// TIA Portal V18 export
FUNCTION "ST10Cyl_interface81-90" : Void   // FC1028, LAD
{ S7_Optimized_Access := 'FALSE' }
VERSION : 0.1
// stored: AutoNumber false, IsIECCheckEnabled false, SetENOAutomatically false, UDAEnableTagReadback false
   VAR_INPUT
      AlwaysON : Bool;
      E_stop : Bool;
   END_VAR
   VAR_TEMP
      tTest : Bool;
   END_VAR
BEGIN

REGION Network 1 (SCL): Cylinder 81-90 IO Interface (SCL)
   (*
   //Cylinder81 IO  L-UnloadingTransCylinder
   //Input
   "ST10Cylinder".Cy[81].In.WorkPositionSensor := "iL-UnloadingTransCylinderInWP";
   "ST10Cylinder".Cy[81].In.HomePositionSensor := "iL-UnloadingTransCylinderInHP";
   //Output
   "oL-UnloadingTransCylinderToWP" := "ST10Cylinder".Cy[81].Out.GoWorkPosition;
   "oL-UnloadingTransCylinderToHP" := "ST10Cylinder".Cy[81].Out.GoHomePosition;

   //Cylinder82 IO  L-UnloadingTransPalletLocationCylinder
   //Input
   "ST10Cylinder".Cy[82].In.WorkPositionSensor := "iL-UnloadingTransPalletLocationCylinderInWP";
   "ST10Cylinder".Cy[82].In.HomePositionSensor := "iL-UnloadingTransPalletLocationCylinderInHP";
   //Output
   "oL-UnloadingTransPalletLocationCylinderToWP" := "ST10Cylinder".Cy[82].Out.GoWorkPosition;
   "oL-UnloadingTransPalletLocationCylinderToHP" := "ST10Cylinder".Cy[82].Out.GoHomePosition;

   //Cylinder83 IO  L-UnloadingStopperCylinder1_1
   //Input
   "ST10Cylinder".Cy[83].In.WorkPositionSensor := "oL-UnloadingStopperCylinder1_1";
   "ST10Cylinder".Cy[83].In.HomePositionSensor := NOT "oL-UnloadingStopperCylinder1_1";
   //Output
   "oL-UnloadingStopperCylinder1_1" := "ST10Cylinder".Cy[83].Out.GoWorkPosition;
   //"oI-0030TrayLoading8trayStopperCylinderToHP" := "ST10Cylinder".Cy[83].Out.GoHomePosition;

   //Cylinder84 IO  L-UnloadingStopperCylinder1_2
   //Input
   "ST10Cylinder".Cy[84].In.WorkPositionSensor := "oL-UnloadingStopperCylinder1_2";
   "ST10Cylinder".Cy[84].In.HomePositionSensor := NOT "oL-UnloadingStopperCylinder1_2";
   //Output
   "oL-UnloadingStopperCylinder1_2" := "ST10Cylinder".Cy[84].Out.GoWorkPosition;
   //"oI-0080TrayLoadingTaketrayCylinderToHP" := "ST10Cylinder".Cy[84].Out.GoHomePosition;

   //Cylinder85 IO  L-UnloadingStopperCylinder2_1
   //Input
   "ST10Cylinder".Cy[85].In.WorkPositionSensor := "oL-UnloadingStopperCylinder2_1";
   "ST10Cylinder".Cy[85].In.HomePositionSensor := NOT "oL-UnloadingStopperCylinder2_1";
   //Output
   "oL-UnloadingStopperCylinder2_1" := "ST10Cylinder".Cy[85].Out.GoWorkPosition;
   //"oI-0050TrayLoadingTrayCylinderToHP" := "ST10Cylinder".Cy[85].Out.GoHomePosition;

   //Cylinder86  L-UnloadingStopperCylinder2_2
   //Input
   "ST10Cylinder".Cy[86].In.WorkPositionSensor := "oL-UnloadingStopperCylinder2_2";
   "ST10Cylinder".Cy[86].In.HomePositionSensor := NOT "oL-UnloadingStopperCylinder2_2";
   //Output
   "oL-UnloadingStopperCylinder2_2" := "ST10Cylinder".Cy[86].Out.GoWorkPosition;
   //"oI-0080TrayLoadingTraySupportCylinder1ToHP" := "ST10Cylinder".Cy[86].Out.GoHomePosition;

   //Cylinder87 L-UnloadingStopperCylinder3_1
   //Input
   "ST10Cylinder".Cy[87].In.WorkPositionSensor := "oL-UnloadingStopperCylinder3_1";
   "ST10Cylinder".Cy[87].In.HomePositionSensor := NOT "oL-UnloadingStopperCylinder3_1";
   //Output
   "oL-UnloadingStopperCylinder3_1" := "ST10Cylinder".Cy[87].Out.GoWorkPosition;
   //"oI-0070TrayLoadingTraySupportCylinder8ToHP" := "ST10Cylinder".Cy[87].Out.GoHomePosition;

   //Cylinder88 L-UnloadingStopperCylinder3_2
   //Input
   "ST10Cylinder".Cy[88].In.WorkPositionSensor := "oL-UnloadingStopperCylinder3_2";
   "ST10Cylinder".Cy[88].In.HomePositionSensor := NOT "oL-UnloadingStopperCylinder3_2";
   //Output
   "oL-UnloadingStopperCylinder3_2" := "ST10Cylinder".Cy[88].Out.GoWorkPosition;
   //"oI-0080TrayLoadingTrayLocationCylinderToHP" := "ST10Cylinder".Cy[88].Out.GoHomePosition;
   //
   *)
   (*
   //Cylinder89 K-reserveLoadingStopperCylinder4_1
   //Input
   "ST10Cylinder".Cy[89].In.WorkPositionSensor := "oK-reserveLoadingStopperCylinder4_1";
   "ST10Cylinder".Cy[89].In.HomePositionSensor := NOT "oK-reserveLoadingStopperCylinder4_1";
   //Output
   "oK-reserveLoadingStopperCylinder4_1" := "ST10Cylinder".Cy[89].Out.GoWorkPosition;
   //"oI-0090TrayLoadingTrayUnloadingLiftingCylinderToHP" := "ST10Cylinder".Cy[89].Out.GoHomePosition;

   //Cylinder70 K-reserveLoadingStopperCylinder4_2
   // //Input
   "ST10Cylinder".Cy[70].In.WorkPositionSensor := "oK-reserveLoadingStopperCylinder4_2";
   "ST10Cylinder".Cy[70].In.HomePositionSensor := NOT "oK-reserveLoadingStopperCylinder4_2";
   // //Output
   "oK-reserveLoadingStopperCylinder4_2" := "ST10Cylinder".Cy[70].Out.GoWorkPosition;
   // "Feeding washer  lift Cylinder ToHP" := "ST10Cylinder".Cy[70].Out.GoHomePosition;

   *)
END_REGION

REGION Network 2: CY81 interface L-UnloadingTransCylinder
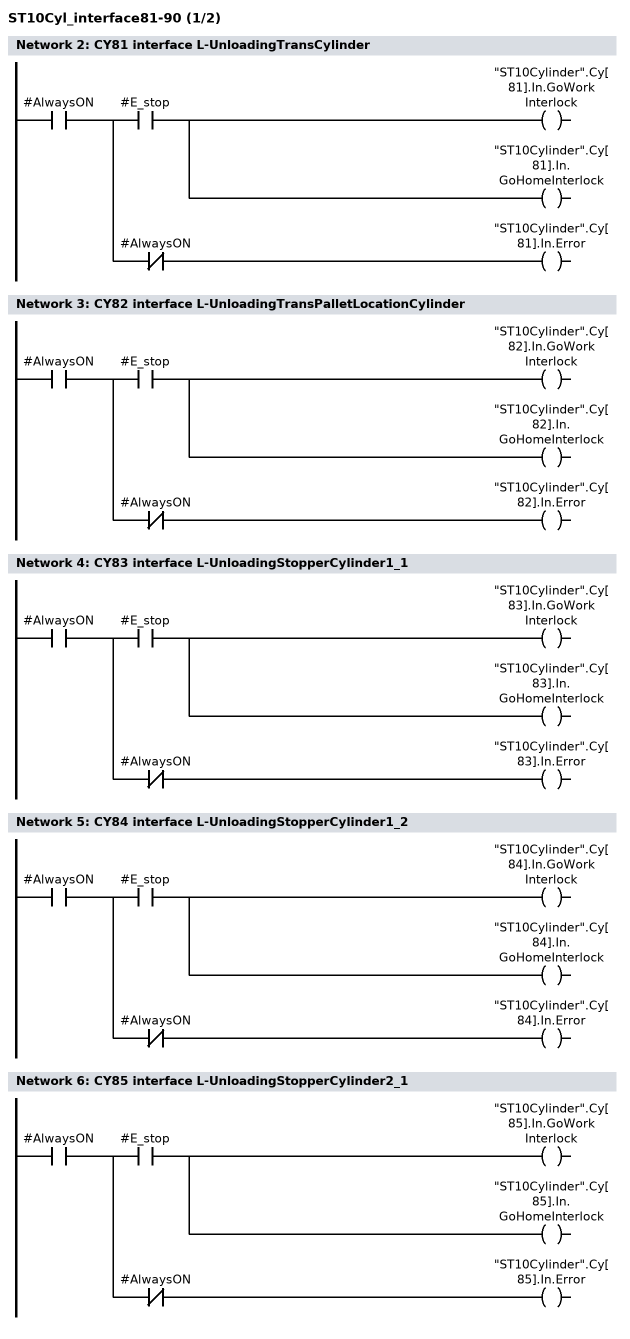
   RUNG wire#powerrail
      Contact( #AlwaysON )
      wire#w1
      Contact( #E_stop )
      wire#w2
      Coil( "ST10Cylinder".Cy[81].In.GoWorkInterlock )
   END_RUNG
   RUNG wire#w2
      Coil( "ST10Cylinder".Cy[81].In.GoHomeInterlock )
   END_RUNG
   RUNG wire#w1
      I_Contact( #AlwaysON )
      Coil( "ST10Cylinder".Cy[81].In.Error )
   END_RUNG
   // the same network as SCL:
   "ST10Cylinder".Cy[81].In.GoWorkInterlock := #AlwaysON AND #E_stop;
   "ST10Cylinder".Cy[81].In.GoHomeInterlock := #AlwaysON AND #E_stop;
   "ST10Cylinder".Cy[81].In.Error := #AlwaysON AND NOT #AlwaysON;
END_REGION

REGION Network 3: CY82 interface L-UnloadingTransPalletLocationCylinder
   RUNG wire#powerrail
      Contact( #AlwaysON )
      wire#w1
      Contact( #E_stop )
      wire#w2
      Coil( "ST10Cylinder".Cy[82].In.GoWorkInterlock )
   END_RUNG
   RUNG wire#w2
      Coil( "ST10Cylinder".Cy[82].In.GoHomeInterlock )
   END_RUNG
   RUNG wire#w1
      I_Contact( #AlwaysON )
      Coil( "ST10Cylinder".Cy[82].In.Error )
   END_RUNG
   // the same network as SCL:
   "ST10Cylinder".Cy[82].In.GoWorkInterlock := #AlwaysON AND #E_stop;
   "ST10Cylinder".Cy[82].In.GoHomeInterlock := #AlwaysON AND #E_stop;
   "ST10Cylinder".Cy[82].In.Error := #AlwaysON AND NOT #AlwaysON;
END_REGION

REGION Network 4: CY83 interface L-UnloadingStopperCylinder1_1
   RUNG wire#powerrail
      Contact( #AlwaysON )
      wire#w1
      Contact( #E_stop )
      wire#w2
      Coil( "ST10Cylinder".Cy[83].In.GoWorkInterlock )
   END_RUNG
   RUNG wire#w2
      Coil( "ST10Cylinder".Cy[83].In.GoHomeInterlock )
   END_RUNG
   RUNG wire#w1
      I_Contact( #AlwaysON )
      Coil( "ST10Cylinder".Cy[83].In.Error )
   END_RUNG
   // the same network as SCL:
   "ST10Cylinder".Cy[83].In.GoWorkInterlock := #AlwaysON AND #E_stop;
   "ST10Cylinder".Cy[83].In.GoHomeInterlock := #AlwaysON AND #E_stop;
   "ST10Cylinder".Cy[83].In.Error := #AlwaysON AND NOT #AlwaysON;
END_REGION

REGION Network 5: CY84 interface L-UnloadingStopperCylinder1_2
   RUNG wire#powerrail
      Contact( #AlwaysON )
      wire#w1
      Contact( #E_stop )
      wire#w2
      Coil( "ST10Cylinder".Cy[84].In.GoWorkInterlock )
   END_RUNG
   RUNG wire#w2
      Coil( "ST10Cylinder".Cy[84].In.GoHomeInterlock )
   END_RUNG
   RUNG wire#w1
      I_Contact( #AlwaysON )
      Coil( "ST10Cylinder".Cy[84].In.Error )
   END_RUNG
   // the same network as SCL:
   "ST10Cylinder".Cy[84].In.GoWorkInterlock := #AlwaysON AND #E_stop;
   "ST10Cylinder".Cy[84].In.GoHomeInterlock := #AlwaysON AND #E_stop;
   "ST10Cylinder".Cy[84].In.Error := #AlwaysON AND NOT #AlwaysON;
END_REGION

REGION Network 6: CY85 interface L-UnloadingStopperCylinder2_1
   RUNG wire#powerrail
      Contact( #AlwaysON )
      wire#w1
      Contact( #E_stop )
      wire#w2
      Coil( "ST10Cylinder".Cy[85].In.GoWorkInterlock )
   END_RUNG
   RUNG wire#w2
      Coil( "ST10Cylinder".Cy[85].In.GoHomeInterlock )
   END_RUNG
   RUNG wire#w1
      I_Contact( #AlwaysON )
      Coil( "ST10Cylinder".Cy[85].In.Error )
   END_RUNG
   // the same network as SCL:
   "ST10Cylinder".Cy[85].In.GoWorkInterlock := #AlwaysON AND #E_stop;
   "ST10Cylinder".Cy[85].In.GoHomeInterlock := #AlwaysON AND #E_stop;
   "ST10Cylinder".Cy[85].In.Error := #AlwaysON AND NOT #AlwaysON;
END_REGION

REGION Network 7: CY86 interface L-UnloadingStopperCylinder2_2
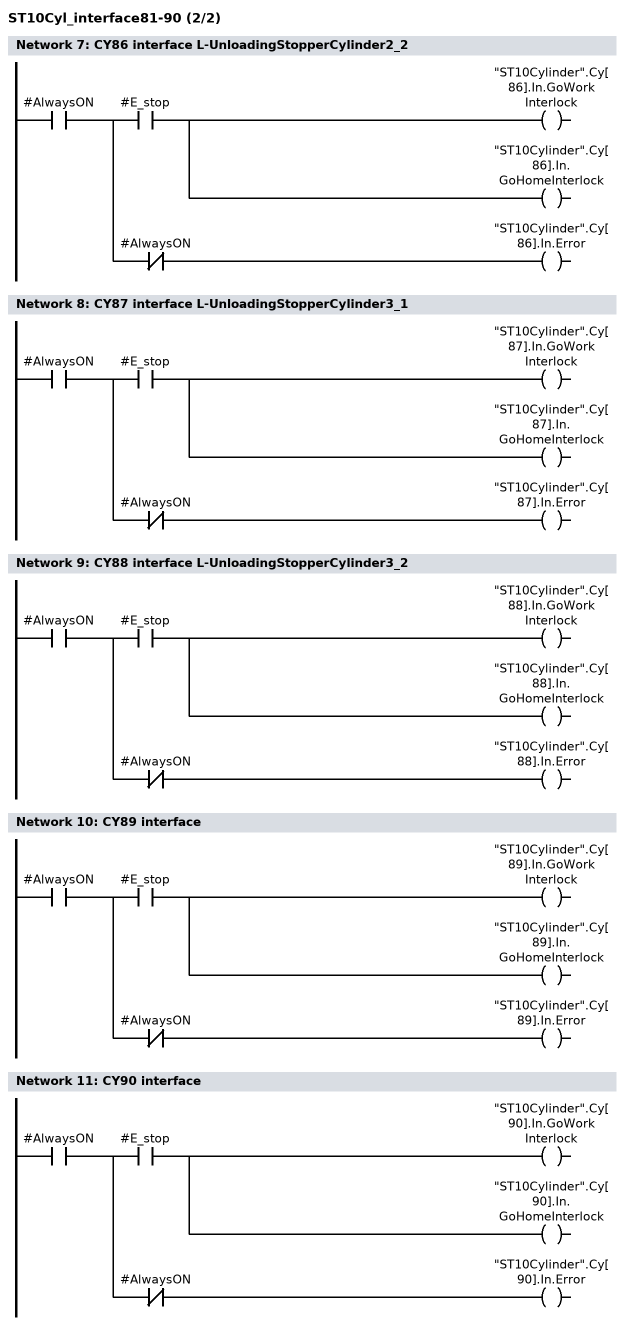
   RUNG wire#powerrail
      Contact( #AlwaysON )
      wire#w1
      Contact( #E_stop )
      wire#w2
      Coil( "ST10Cylinder".Cy[86].In.GoWorkInterlock )
   END_RUNG
   RUNG wire#w2
      Coil( "ST10Cylinder".Cy[86].In.GoHomeInterlock )
   END_RUNG
   RUNG wire#w1
      I_Contact( #AlwaysON )
      Coil( "ST10Cylinder".Cy[86].In.Error )
   END_RUNG
   // the same network as SCL:
   "ST10Cylinder".Cy[86].In.GoWorkInterlock := #AlwaysON AND #E_stop;
   "ST10Cylinder".Cy[86].In.GoHomeInterlock := #AlwaysON AND #E_stop;
   "ST10Cylinder".Cy[86].In.Error := #AlwaysON AND NOT #AlwaysON;
END_REGION

REGION Network 8: CY87 interface L-UnloadingStopperCylinder3_1
   RUNG wire#powerrail
      Contact( #AlwaysON )
      wire#w1
      Contact( #E_stop )
      wire#w2
      Coil( "ST10Cylinder".Cy[87].In.GoWorkInterlock )
   END_RUNG
   RUNG wire#w2
      Coil( "ST10Cylinder".Cy[87].In.GoHomeInterlock )
   END_RUNG
   RUNG wire#w1
      I_Contact( #AlwaysON )
      Coil( "ST10Cylinder".Cy[87].In.Error )
   END_RUNG
   // the same network as SCL:
   "ST10Cylinder".Cy[87].In.GoWorkInterlock := #AlwaysON AND #E_stop;
   "ST10Cylinder".Cy[87].In.GoHomeInterlock := #AlwaysON AND #E_stop;
   "ST10Cylinder".Cy[87].In.Error := #AlwaysON AND NOT #AlwaysON;
END_REGION

REGION Network 9: CY88 interface L-UnloadingStopperCylinder3_2
   RUNG wire#powerrail
      Contact( #AlwaysON )
      wire#w1
      Contact( #E_stop )
      wire#w2
      Coil( "ST10Cylinder".Cy[88].In.GoWorkInterlock )
   END_RUNG
   RUNG wire#w2
      Coil( "ST10Cylinder".Cy[88].In.GoHomeInterlock )
   END_RUNG
   RUNG wire#w1
      I_Contact( #AlwaysON )
      Coil( "ST10Cylinder".Cy[88].In.Error )
   END_RUNG
   // the same network as SCL:
   "ST10Cylinder".Cy[88].In.GoWorkInterlock := #AlwaysON AND #E_stop;
   "ST10Cylinder".Cy[88].In.GoHomeInterlock := #AlwaysON AND #E_stop;
   "ST10Cylinder".Cy[88].In.Error := #AlwaysON AND NOT #AlwaysON;
END_REGION

REGION Network 10: CY89 interface
   RUNG wire#powerrail
      Contact( #AlwaysON )
      wire#w1
      Contact( #E_stop )
      wire#w2
      Coil( "ST10Cylinder".Cy[89].In.GoWorkInterlock )
   END_RUNG
   RUNG wire#w2
      Coil( "ST10Cylinder".Cy[89].In.GoHomeInterlock )
   END_RUNG
   RUNG wire#w1
      I_Contact( #AlwaysON )
      Coil( "ST10Cylinder".Cy[89].In.Error )
   END_RUNG
   // the same network as SCL:
   "ST10Cylinder".Cy[89].In.GoWorkInterlock := #AlwaysON AND #E_stop;
   "ST10Cylinder".Cy[89].In.GoHomeInterlock := #AlwaysON AND #E_stop;
   "ST10Cylinder".Cy[89].In.Error := #AlwaysON AND NOT #AlwaysON;
END_REGION

REGION Network 11: CY90 interface
   RUNG wire#powerrail
      Contact( #AlwaysON )
      wire#w1
      Contact( #E_stop )
      wire#w2
      Coil( "ST10Cylinder".Cy[90].In.GoWorkInterlock )
   END_RUNG
   RUNG wire#w2
      Coil( "ST10Cylinder".Cy[90].In.GoHomeInterlock )
   END_RUNG
   RUNG wire#w1
      I_Contact( #AlwaysON )
      Coil( "ST10Cylinder".Cy[90].In.Error )
   END_RUNG
   // the same network as SCL:
   "ST10Cylinder".Cy[90].In.GoWorkInterlock := #AlwaysON AND #E_stop;
   "ST10Cylinder".Cy[90].In.GoHomeInterlock := #AlwaysON AND #E_stop;
   "ST10Cylinder".Cy[90].In.Error := #AlwaysON AND NOT #AlwaysON;
END_REGION
END_FUNCTION
